// SIMATIC S7-200 project (STEP 7-Micro/WIN), CPU 221 REL 01.10

SYMBOL_TABLE 用户定义1
启动               M10.0
停止               M10.1
加速               M10.2
减速               M10.3
读频率              M10.4
发送完成             SM4.5
END_SYMBOL_TABLE

ORGANIZATION_BLOCK 主程序:OB1
TITLE=S7-200 PLC 与三垦变频器通信用于自动化生产线
// 
// 本程序基于西门子S7-200 PLC与三垦变频器通过RS485通信实现自动化生产线的电机控制。通过PLC与变频器的无缝协作，系统能够精确控制电机的启动、停止、加速、减速，并实时读取和显示电机的运行速度。该系统旨在提升生产线的自动化水平，确保操作员能够通过人机界面（HMI）方便地监控和调整电机运行状态。
// 通讯协议要求配置数据或传输数据信息带字符时，只使用16进制的ASCII编码传输。
// 并且发送命令均需要提前设置命令信息长度，并将命令字符配置到发送存储块中。
// 电机速度应确保处于最大频率50hz和最小频率15hz之间，确保电机在安全和有效的范围内运行。
// 程序应该确保，在使用HMI的按钮时每次点击仅出发一次指令。
// 
// PLC在开机时，会检测开机状态位，若开机状态正常，则开始做通讯初始化工作，初始化PLC与三垦变频器的通讯协议。
// 在做任何的操作之前，PLC会先检测通信就绪标志位，以此来检查PLC是否已经准备好与变频器进行通信。
// 通讯要求配置数据或传输数据信息带字符时，只使用16进制的ASCII编码传输。
// 本次通讯使用的本地PLC默认站号为'0'；通讯目标是一台三垦变频器，该变频器的站号为'4'。
// 配置通讯的开始符号为星号'*'，以及终止符号为回车符。
// 通讯将最大接收长度限制为14个字节，以及空闲线时间为5ms。
// 配置完成后，PLC将发送缓冲区准备就绪，进入与变频器通信的待命状态。
// 
// 在HMI（人机界面）中分别有一个开启和停止按钮控制变频器的启动或停止操作，当按钮被按下时，PLC应开始相应的给变频器发送启动或停止命令。本次通讯使用的启动命令为字符'P'，停止命令为字符'R'，命令信息长度均为6个字节。
// 发送命令后，PLC通过数据发送完成状态位驱动外部指示灯，及时为用户显示发送完成状态。
// 
// 在HMI中有一个加速按钮、一个减速按钮可以调控变频器的目标频率数值的增加或减少。
// 程序维护一个10ms的时间窗口计时器，用来确保电机的平稳运行，避免电机频率过快变化。
// 当PLC检测到调节电机频率目标值与电机实际速度值不一致时，PLC发送频率调整命令。
// 调节电机频率指令的字符为字符'O'，数据长度为11字节。
// 目标频率需要转换为BCD编码，再转为ASCII格式，最后再存储至发送缓冲区，才能执行发送指令。
// 
// 在HMI中有一个读取电机速度按钮，当读取电机速度的按钮被按下时，PLC应开始发送读取命令。
// 使用的读取命令字符为'C'，命令信息长度为6个字节。
// PLC不断检测接收缓冲区中的数据是否接收到了是读取命令'C'，若检测到读取命令'C'，,PLC将接收缓冲区的数据转换为BCD编码，并存放在显示频率HMI端口中。
// 发送完成进入接收中断。
BEGIN
Network 1
LD     SM0.1
CALL   初始化:SBR0
?000
Network 2
LD     启动:M10.0
EU
MOVB   6, VB100
MOVB   16#50, VB104
CALL   发送:SBR1
Network 3
LDB<>  SMB86, 0
MOVB   SMB86, VB400
Network 4
LD     发送完成:SM4.5
=      Q0.0
Network 5
LD     停止:M10.1
EU
MOVB   6, VB100
MOVB   16#52, VB104
CALL   发送:SBR1
Network 6
LDN    T37
TON    T37, 10
Network 7
LD     加速:M10.2
A      T37
INCW   VW135
Network 8
LD     减速:M10.3
A      T37
DECW   VW135
Network 9
LDW>=  VW135, 50
MOVW   50, VW135
Network 10
LDW<=  VW135, 15
MOVW   15, VW135
Network 11
LDW<>  VW135, VW145
MOVB   11, VB100
MOVB   16#4F, VB104
MOVW   VW135, VW137
IBCD   VW137
MOVW   VW137, VW143
*I     16#10, VW143
HTA    VB143, VB105, 5
MOVW   VW135, VW145
CALL   发送:SBR1
Network 12
LD     读频率:M10.4
EU
MOVB   6, VB100
MOVB   16#43, VB104
CALL   发送:SBR1
Network 13
LDB=   VB204, 16#43
HTA    VB205, VB500, 4
MOVW   VW500, VW600
BCDI   VW600
MOVW   VW600, VW602
/I     +10, VW602
END_ORGANIZATION_BLOCK

SUBROUTINE_BLOCK 初始化:SBR0
TITLE=
BEGIN
Network 1
LD     SM0.0
MOVB   16#9, SMB30
MOVB   16#F0, SMB87
MOVB   16#2A, SMB88
MOVB   16#D, SMB89
MOVB   14, SMB94
MOVW   5, SMW90
Network 2
LD     SM0.0
MOVB   16#2A, VB101
MOVB   16#30, VB102
MOVB   16#34, VB103
Network 3
LD     SM0.0
ATCH   接收中断:INT0, 9
ENI
END_SUBROUTINE_BLOCK

SUBROUTINE_BLOCK 发送:SBR1
TITLE=
BEGIN
Network 1
LD     SM0.0
MOVD   &VB101, VD131
MOVW   0, VW129
MOVB   VB100, AC1
MOVW   AC1, VW127
-I     +2, VW127
Network 2
LD     SM0.0
FOR    VW125, 1, VW127
Network 3
LD     SM0.0
MOVB   *VD131, AC0
+I     AC0, VW129
+D     1, VD131
Network 4
NEXT
Network 5
LD     SM0.0
MOVW   16#FF, AC0
ANDW   VW129, AC0
INVW   AC0
+I     1, AC0
ANDW   16#7F, AC0
ORW    16#40, AC0
MOVB   AC0, *VD131
+D     1, VD131
MOVB   16#D, *VD131
Network 6
LD     SM0.0
XMT    VB100, 0
Network 7
LD     SM0.0
CRET
END_SUBROUTINE_BLOCK

INTERRUPT_BLOCK 接收中断:INT0
TITLE=
BEGIN
Network 1
LD     SM0.0
RCV    VB200, 0
END_INTERRUPT_BLOCK
